(* Logix 5000 project; controller STAT 1756-L72 rev 20.12; software revision 20.04; part 9 of 34 *)
(* tags used below, declared in another part *)
   B14 : DINT[30];
   B16 : DINT[30];
   B17 : DINT[30];
   B3 : DINT[256];
   DateTime : DINT[7];   // DINT array tag for retrieve wallclock time through GSV created during conversion
   I10_000_Bit07 : ALIAS FOR I10[0].7;   // Hand Automaat CL8
   I10_000_Bit10 : ALIAS FOR I10[0].10;   // Drukknop start CL8 PM1
   I10_000_Bit11 : ALIAS FOR I10[0].11;   // Drukknop stop CL8 PM1
   I10_000_Bit12 : ALIAS FOR I10[0].12;   // Drukknop start CL8 PM2
   I10_000_Bit13 : ALIAS FOR I10[0].13;   // Drukknop stop CL8 PM2
   I10_000_Bit14 : ALIAS FOR I10[0].14;   // Drukknop start CL8 PM3
   I10_000_Bit15 : ALIAS FOR I10[0].15;   // Drukknop stop CL8 PM3
   I10_001_Bit00 : ALIAS FOR I10[1].0;   // Drukknop start CL8 PM4
   I10_001_Bit01 : ALIAS FOR I10[1].1;   // Drukknop stop CL8 PM4
   I1_016_Bit02 : ALIAS FOR I1[16].2;   // CL2 start p11
   I1_016_Bit03 : ALIAS FOR I1[16].3;   // CL2 stop p11
   I1_016_Bit04 : ALIAS FOR I1[16].4;   // CL2 start p12
   I1_016_Bit05 : ALIAS FOR I1[16].5;   // CL2 stop p12
   I1_016_Bit11 : ALIAS FOR I1[16].11;   // Niveau lus5 kontakt1
   I1_016_Bit12 : ALIAS FOR I1[16].12;   // Niveau lus5 kontakt2
   I1_017_Bit02 : ALIAS FOR I1[17].2;   // CL3 start p13
   I1_017_Bit03 : ALIAS FOR I1[17].3;   // CL3 stop p13
   I1_017_Bit04 : ALIAS FOR I1[17].4;   // CL3 start p14
   I1_017_Bit05 : ALIAS FOR I1[17].5;   // CL3 stop p14
   I1_017_Bit11 : ALIAS FOR I1[17].11;   // Niveau lus6 kontakt1
   I1_017_Bit12 : ALIAS FOR I1[17].12;   // Niveau lus6 kontakt2
   I1_018_Bit02 : ALIAS FOR I1[18].2;   // CL4 start p15
   I1_018_Bit03 : ALIAS FOR I1[18].3;   // CL4 stop p15
   I1_018_Bit04 : ALIAS FOR I1[18].4;   // CL4 start p16
   I1_018_Bit05 : ALIAS FOR I1[18].5;   // CL4 stop p16
   I1_018_Bit11 : ALIAS FOR I1[18].11;   // Niveau lus7 kontakt1
   I1_018_Bit12 : ALIAS FOR I1[18].12;   // Niveau lus7 kontakt2
   I1_018_Bit13 : ALIAS FOR I1[18].13;   // Niveau lus7 kontakt3
   I2_000_Bit00 : ALIAS FOR I2[0].0;   // Deelnoodstop cl2 lijn 1
   I2_000_Bit01 : ALIAS FOR I2[0].1;   // Deelnoodstop cl3 lijn 3
   I2_000_Bit02 : ALIAS FOR I2[0].2;   // Deelnoodstop cl4
   I2_000_Bit03 : ALIAS FOR I2[0].3;   // Deelnoodstop cl5 lijn 4
   I2_000_Bit06 : ALIAS FOR I2[0].6;   // Deelnoodstop cl7 IBT B
   I6_001_Bit12 : ALIAS FOR I6[1].12;   // Ph meting vervuild water fout
   I7_000_Bit01 : ALIAS FOR I7[0].1;   // lus2 niveau kontakt 1
   I7_000_Bit04 : ALIAS FOR I7[0].4;   // lus3 niveau kontakt 1
   I7_000_Bit10 : ALIAS FOR I7[0].10;   // zeer hoog alarm ketel clarifee
   I7_001_Bit13 : ALIAS FOR I7[1].13;   // lus 8 niveau kontakt 1
   I7_001_Bit14 : ALIAS FOR I7[1].14;   // lus 8 niveau kontakt 2
   I7_001_Bit15 : ALIAS FOR I7[1].15;   // lus 8 niveau kontakt 3
   I8_001_Bit01 : ALIAS FOR I8[1].1;   // hand automaat cl5
   I8_001_Bit02 : ALIAS FOR I8[1].2;   // drukknop start cl5 p17
   I8_001_Bit03 : ALIAS FOR I8[1].3;   // drukknop stop cl5 p17
   I8_001_Bit04 : ALIAS FOR I8[1].4;   // drukknop start cl5 p18
   I8_001_Bit05 : ALIAS FOR I8[1].5;   // drukknop stop cl5 p18
   I9_000_Bit09 : ALIAS FOR I9[0].9;   // Hand_Auto CL7
   I9_001_Bit12 : ALIAS FOR I9[1].12;   // Drukknop start CL7 A
   I9_001_Bit13 : ALIAS FOR I9[1].13;   // Drukknop stop CL7 pd7
   I9_001_Bit14 : ALIAS FOR I9[1].14;   // drukknop start cl7 pd8
   I9_001_Bit15 : ALIAS FOR I9[1].15;   // drukknop stop cl7 pd8
   N11 : DINT[150];
   N12 : DINT[230];
   N13 : DINT[230];
   N20 : DINT[80];
   N21 : DINT[80];
   O12_000_Bit04 : ALIAS FOR O12[0].4;   // Motor doseerpomp acide pd3 PD3_DOS_ACIDE
   O12_000_Bit05 : ALIAS FOR O12[0].5;   // Motor doseerpomp acide pd4 PD4_DOS_ACIDE
   O12_000_Bit06 : ALIAS FOR O12[0].6;   // Motor doseerpomp acide pd5 soude PD5_DOS_SOUDE
   O12_000_Bit07 : ALIAS FOR O12[0].7;   // Motor doseerpomp acide pd6 soude PD6_DOS_SOUDE
   O12_000_Bit10 : ALIAS FOR O12[0].10;   // pomp pd7 doseerpomp floculaat PD7_DOSEER_FLOCU
   O12_000_Bit11 : ALIAS FOR O12[0].11;   // pomp pd8 doseerpomp floculaat PD8_DOSEER_FLOCU
   O12_000_Bit14 : ALIAS FOR O12[0].14;   // Motor Pm1 recerculatiepomp ingang 1 decanter PM1_RECER_DEC1
   O12_000_Bit15 : ALIAS FOR O12[0].15;   // Motor Pm2 recerculatiepomp ingang 2 decanter PM2_RECER_DEC2
   O12_001_Bit00 : ALIAS FOR O12[1].0;   // Motor Pm3 evacuatiepomp ingang 1 decanter PM3_EVACU_IN_1
   O12_001_Bit01 : ALIAS FOR O12[1].1;   // Motor Pm4 evacuatiepomp ingang 2 decanter PM4_EVACU_IN_2
   O13_000_Bit06 : ALIAS FOR O13[0].6;   // PULS_DOSEER_PD3
   O13_000_Bit07 : ALIAS FOR O13[0].7;   // PULS_DOSEER_PD4
   O13_000_Bit08 : ALIAS FOR O13[0].8;   // PULS_DOSEER_PD5
   O13_000_Bit09 : ALIAS FOR O13[0].9;   // PULS_DOSEER_PD6
   O15_001_Bit07 : ALIAS FOR O15[1].7;   // EV3 EV3
   O15_001_Bit08 : ALIAS FOR O15[1].8;   // EV4 EV4
   O15_001_Bit09 : ALIAS FOR O15[1].9;   // EV5 EV5
   P11_RECUP : BOOL;
   P13_RECUP : BOOL;
   P14_RECUP : BOOL;
   p15 : BOOL;
   P16 : BOOL;
   P17 : BOOL;
   P18 : BOOL;
   pd3 : BOOL;
   pd4 : BOOL;
   pd5 : BOOL;
   pd6 : BOOL;
   PD7 : BOOL;
   PD8 : BOOL;
   PM1 : BOOL;
   PM2 : BOOL;
   PM3 : BOOL;
   PM4 : BOOL;
   PMP_L1_ET_L3_RUN : BOOL;
   POS_EV3 : BOOL;
   T27 : TIMER[100];
   T4 : TIMER[200];
(* ibt, continued *)

ROUTINE _11_PM1_PM4   (* ladder *)
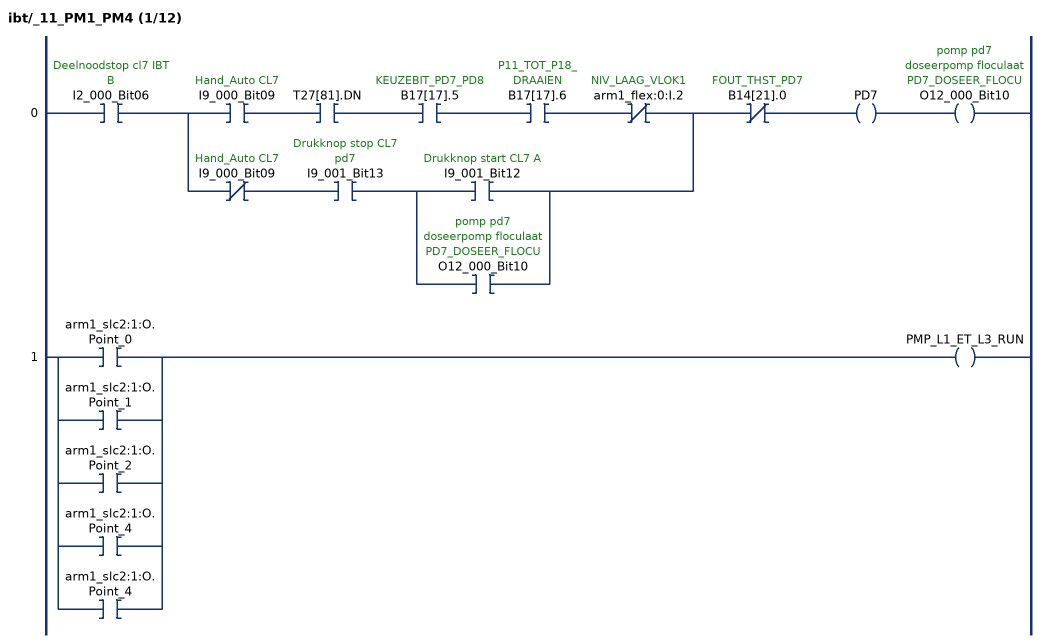
   0: XIC(I2_000_Bit06)[XIC(I9_000_Bit09) XIC(T27[81].DN) XIC(B17[17].5) XIC(B17[17].6) XIO(arm1_flex:0:I.2) ,XIO(I9_000_Bit09) XIC(I9_001_Bit13) [XIC(I9_001_Bit12) ,XIC(O12_000_Bit10) ] ]XIO(B14[21].0)OTE(PD7)OTE(O12_000_Bit10);
   1: [XIC(arm1_slc2:1:O.Point_0) ,[XIC(arm1_slc2:1:O.Point_1) ,[XIC(arm1_slc2:1:O.Point_2) ,[XIC(arm1_slc2:1:O.Point_4) ,XIC(arm1_slc2:1:O.Point_4) ] ] ] ]OTE(PMP_L1_ET_L3_RUN);
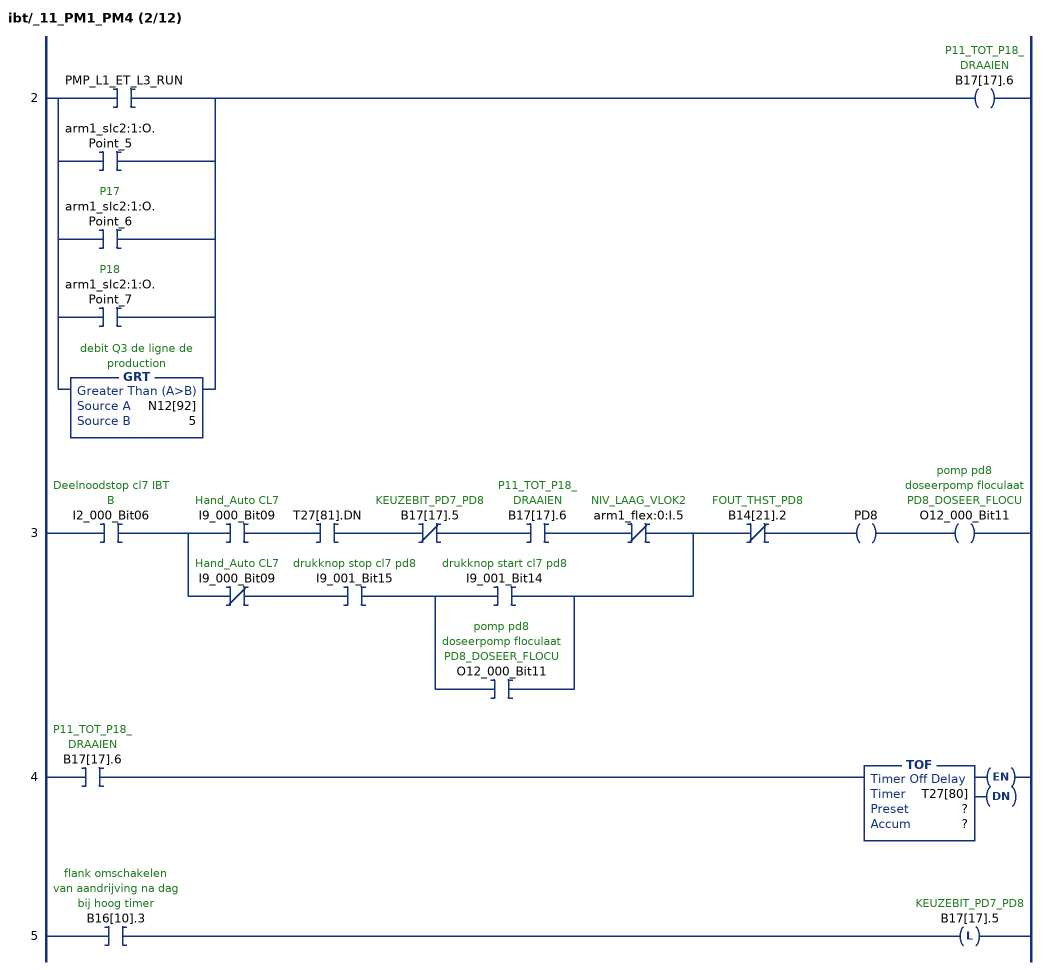
   2: [XIC(PMP_L1_ET_L3_RUN) ,[XIC(arm1_slc2:1:O.Point_5) ,[XIC(arm1_slc2:1:O.Point_6) ,[XIC(arm1_slc2:1:O.Point_7) ,GRT(N12[92],5) ] ] ] ]OTE(B17[17].6);
   3: XIC(I2_000_Bit06)[XIC(I9_000_Bit09) XIC(T27[81].DN) XIO(B17[17].5) XIC(B17[17].6) XIO(arm1_flex:0:I.5) ,XIO(I9_000_Bit09) XIC(I9_001_Bit15) [XIC(I9_001_Bit14) ,XIC(O12_000_Bit11) ] ]XIO(B14[21].2)OTE(PD8)OTE(O12_000_Bit11);
   4: XIC(B17[17].6)TOF(T27[80],?,?);
   5: XIC(B16[10].3)OTL(B17[17].5);
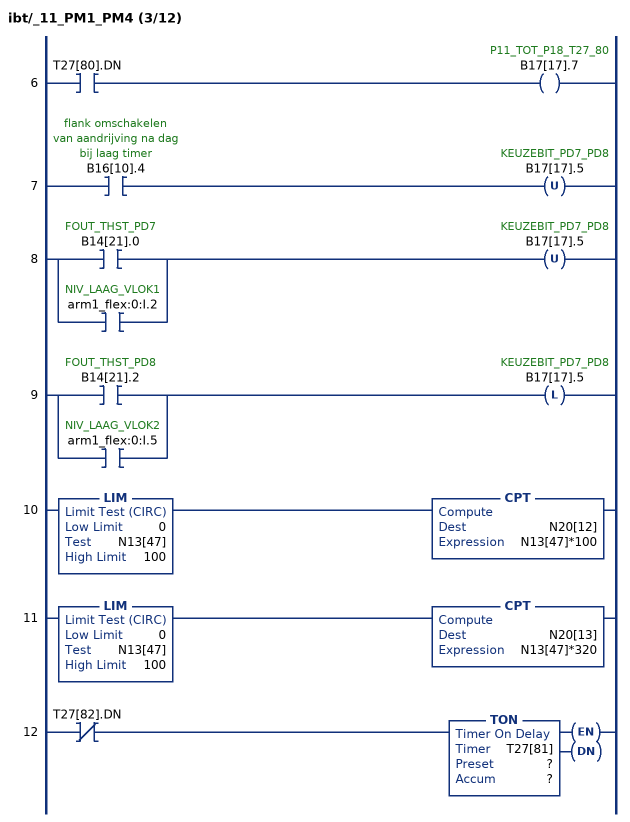
   6: XIC(T27[80].DN)OTE(B17[17].7);
   7: XIC(B16[10].4)OTU(B17[17].5);
   8: [XIC(B14[21].0) ,XIC(arm1_flex:0:I.2) ]OTU(B17[17].5);
   9: [XIC(B14[21].2) ,XIC(arm1_flex:0:I.5) ]OTL(B17[17].5);
   10: LIM(0,N13[47],100)CPT(N20[12],N13[47]*100);
   11: LIM(0,N13[47],100)CPT(N20[13],N13[47]*320);
   12: XIO(T27[82].DN)TON(T27[81],?,?);
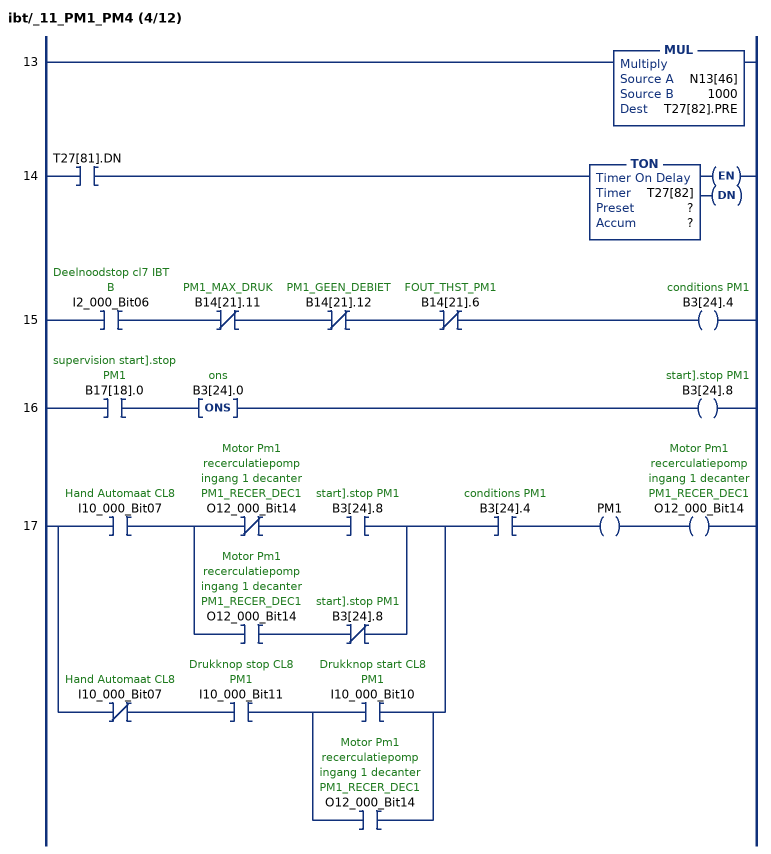
   13: MUL(N13[46],1000,T27[82].PRE);
   14: XIC(T27[81].DN)TON(T27[82],?,?);
   15: XIC(I2_000_Bit06)XIO(B14[21].11)XIO(B14[21].12)XIO(B14[21].6)OTE(B3[24].4);
   16: XIC(B17[18].0)ONS(B3[24].0)OTE(B3[24].8);
   17: [XIC(I10_000_Bit07) [XIO(O12_000_Bit14) XIC(B3[24].8) ,XIC(O12_000_Bit14) XIO(B3[24].8) ] ,XIO(I10_000_Bit07) XIC(I10_000_Bit11) [XIC(I10_000_Bit10) ,XIC(O12_000_Bit14) ] ]XIC(B3[24].4)OTE(PM1)OTE(O12_000_Bit14);
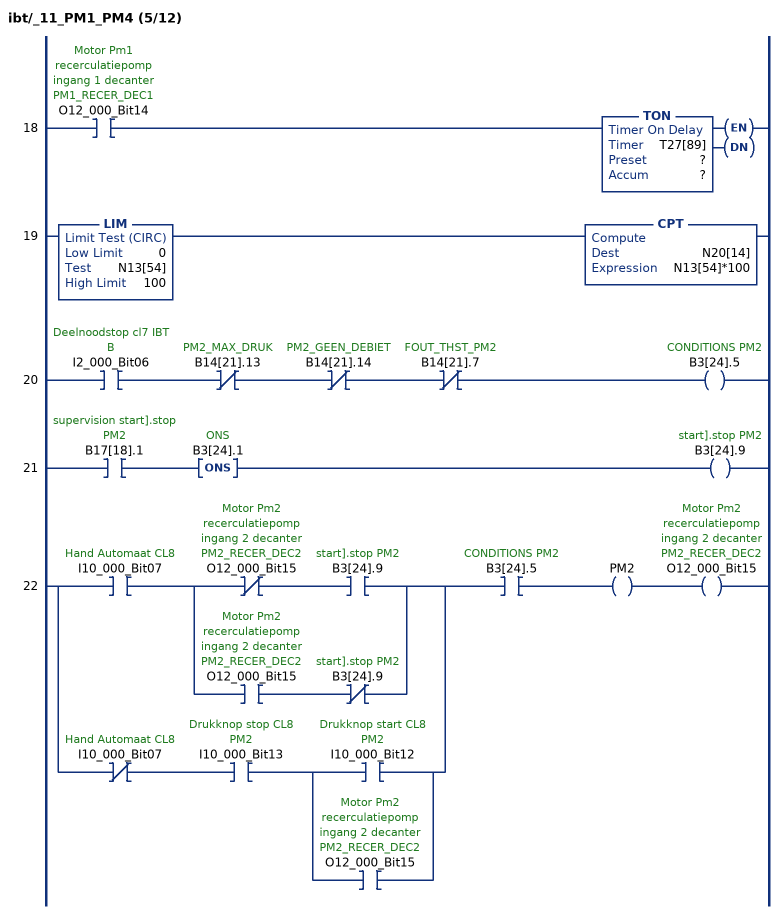
   18: XIC(O12_000_Bit14)TON(T27[89],?,?);
   19: LIM(0,N13[54],100)CPT(N20[14],N13[54]*100);
   20: XIC(I2_000_Bit06)XIO(B14[21].13)XIO(B14[21].14)XIO(B14[21].7)OTE(B3[24].5);
   21: XIC(B17[18].1)ONS(B3[24].1)OTE(B3[24].9);
   22: [XIC(I10_000_Bit07) [XIO(O12_000_Bit15) XIC(B3[24].9) ,XIC(O12_000_Bit15) XIO(B3[24].9) ] ,XIO(I10_000_Bit07) XIC(I10_000_Bit13) [XIC(I10_000_Bit12) ,XIC(O12_000_Bit15) ] ]XIC(B3[24].5)OTE(PM2)OTE(O12_000_Bit15);
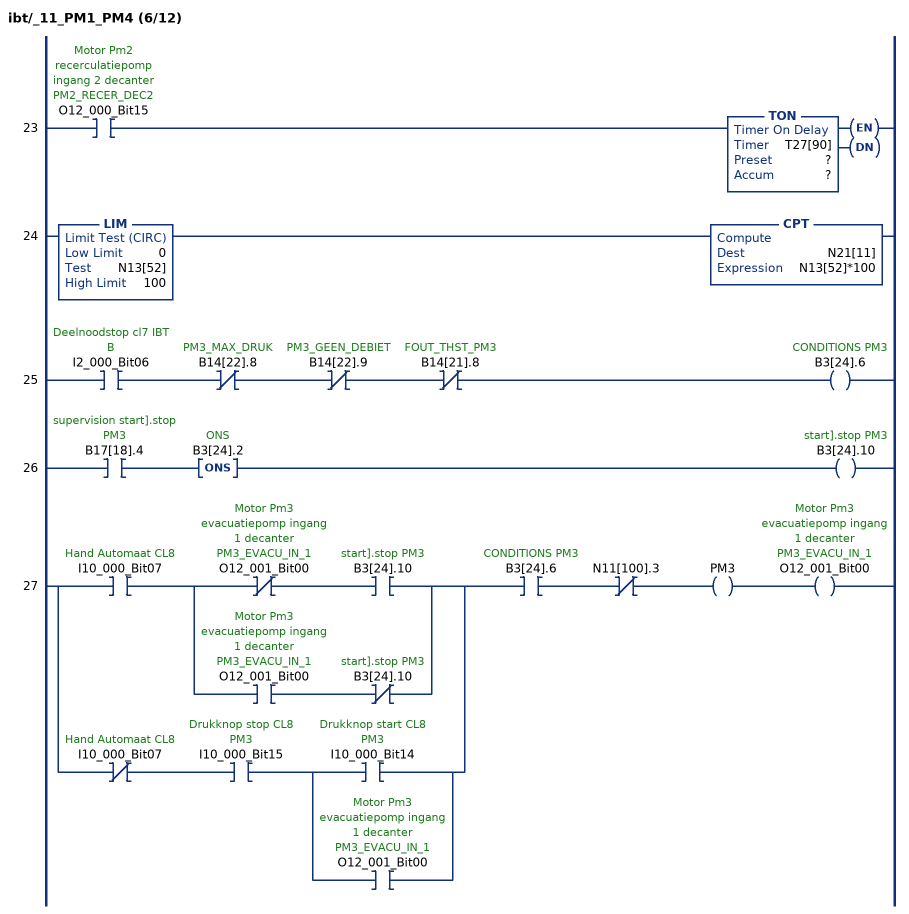
   23: XIC(O12_000_Bit15)TON(T27[90],?,?);
   24: LIM(0,N13[52],100)CPT(N21[11],N13[52]*100);
   25: XIC(I2_000_Bit06)XIO(B14[22].8)XIO(B14[22].9)XIO(B14[21].8)OTE(B3[24].6);
   26: XIC(B17[18].4)ONS(B3[24].2)OTE(B3[24].10);
   27: [XIC(I10_000_Bit07) [XIO(O12_001_Bit00) XIC(B3[24].10) ,XIC(O12_001_Bit00) XIO(B3[24].10) ] ,XIO(I10_000_Bit07) XIC(I10_000_Bit15) [XIC(I10_000_Bit14) ,XIC(O12_001_Bit00) ] ]XIC(B3[24].6)XIO(N11[100].3)OTE(PM3)OTE(O12_001_Bit00);
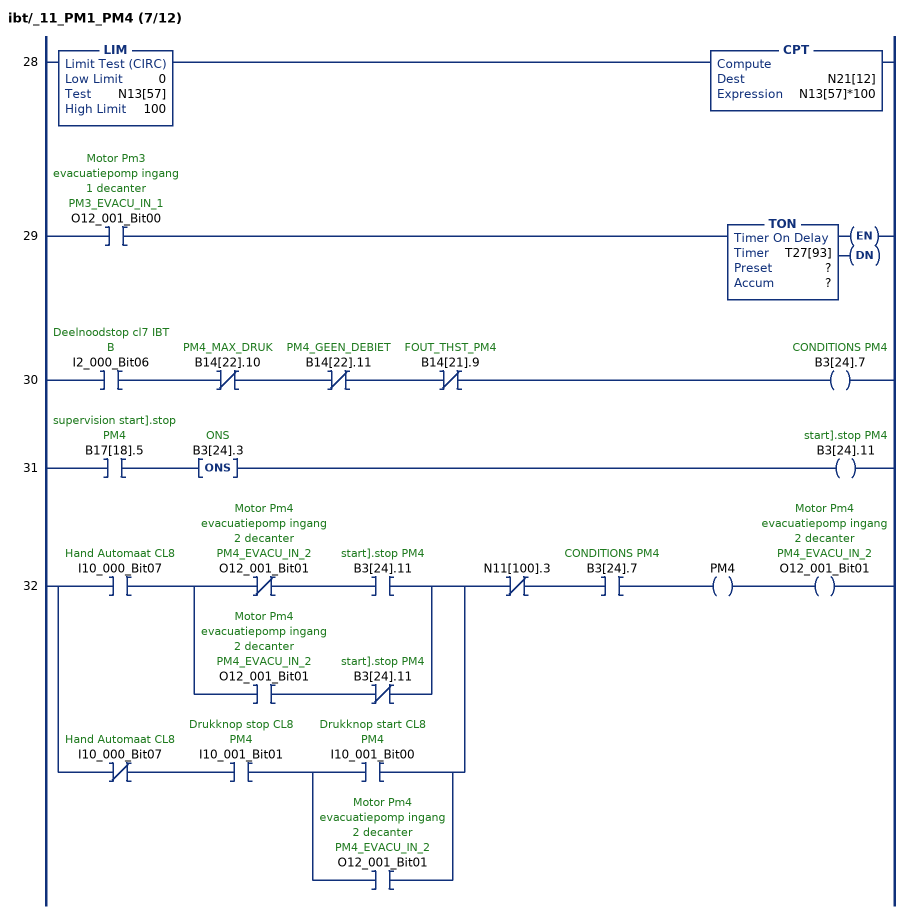
   28: LIM(0,N13[57],100)CPT(N21[12],N13[57]*100);
   29: XIC(O12_001_Bit00)TON(T27[93],?,?);
   30: XIC(I2_000_Bit06)XIO(B14[22].10)XIO(B14[22].11)XIO(B14[21].9)OTE(B3[24].7);
   31: XIC(B17[18].5)ONS(B3[24].3)OTE(B3[24].11);
   32: [XIC(I10_000_Bit07) [XIO(O12_001_Bit01) XIC(B3[24].11) ,XIC(O12_001_Bit01) XIO(B3[24].11) ] ,XIO(I10_000_Bit07) XIC(I10_001_Bit01) [XIC(I10_001_Bit00) ,XIC(O12_001_Bit01) ] ]XIO(N11[100].3)XIC(B3[24].7)OTE(PM4)OTE(O12_001_Bit01);
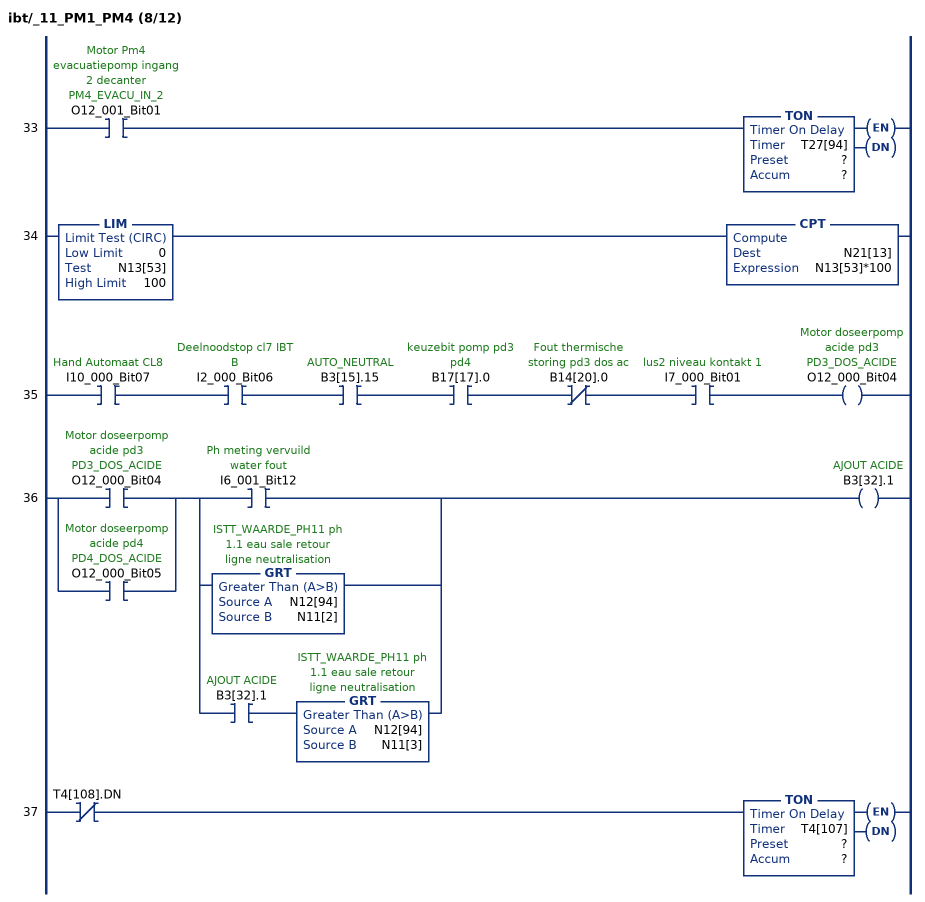
   33: XIC(O12_001_Bit01)TON(T27[94],?,?);
   34: LIM(0,N13[53],100)CPT(N21[13],N13[53]*100);
   35: XIC(I10_000_Bit07)XIC(I2_000_Bit06)XIC(B3[15].15)XIC(B17[17].0)XIO(B14[20].0)XIC(I7_000_Bit01)OTE(O12_000_Bit04);
   36: [XIC(O12_000_Bit04) ,XIC(O12_000_Bit05) ][XIC(I6_001_Bit12) ,GRT(N12[94],N11[2]) ,XIC(B3[32].1) GRT(N12[94],N11[3]) ]OTE(B3[32].1);
   37: XIO(T4[108].DN)TON(T4[107],?,?);
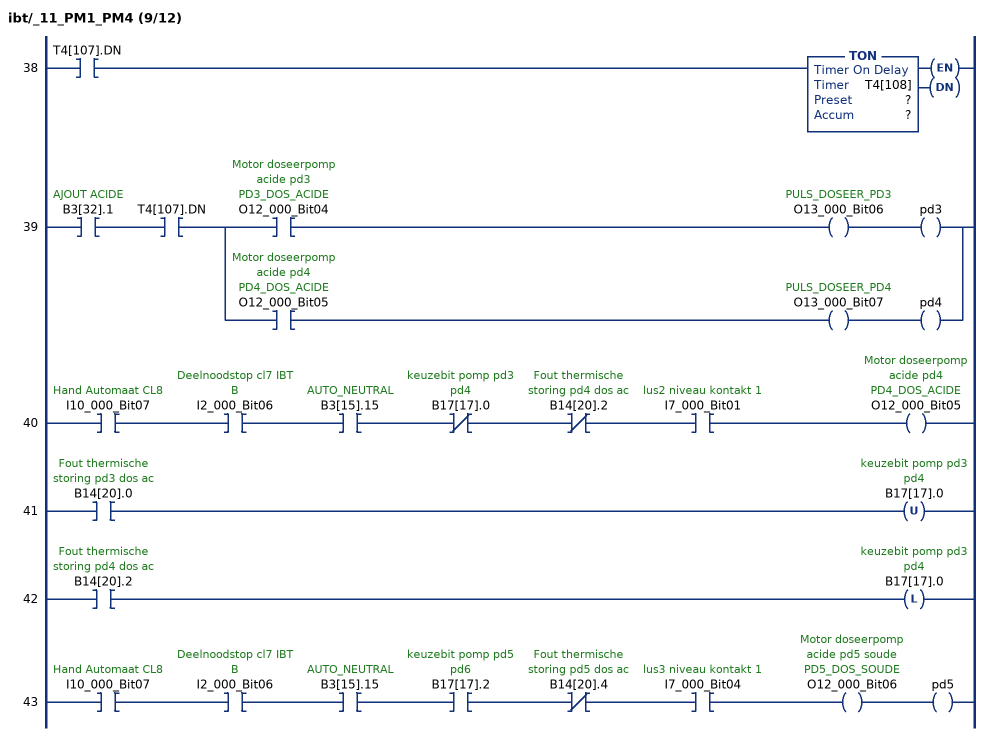
   38: XIC(T4[107].DN)TON(T4[108],?,?);
   39: XIC(B3[32].1)XIC(T4[107].DN)[XIC(O12_000_Bit04) OTE(O13_000_Bit06) OTE(pd3) ,XIC(O12_000_Bit05) OTE(O13_000_Bit07) OTE(pd4) ];
   40: XIC(I10_000_Bit07)XIC(I2_000_Bit06)XIC(B3[15].15)XIO(B17[17].0)XIO(B14[20].2)XIC(I7_000_Bit01)OTE(O12_000_Bit05);
   41: XIC(B14[20].0)OTU(B17[17].0);
   42: XIC(B14[20].2)OTL(B17[17].0);
   43: XIC(I10_000_Bit07)XIC(I2_000_Bit06)XIC(B3[15].15)XIC(B17[17].2)XIO(B14[20].4)XIC(I7_000_Bit04)OTE(O12_000_Bit06)OTE(pd5);
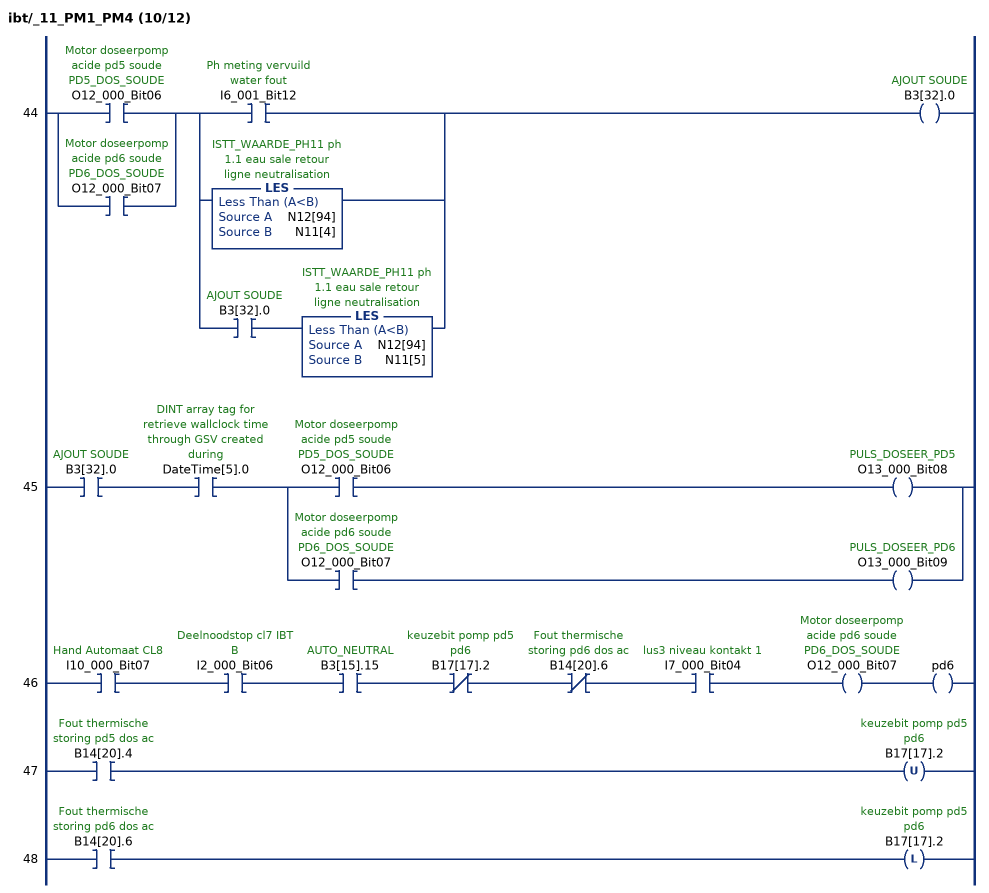
   44: [XIC(O12_000_Bit06) ,XIC(O12_000_Bit07) ][XIC(I6_001_Bit12) ,LES(N12[94],N11[4]) ,XIC(B3[32].0) LES(N12[94],N11[5]) ]OTE(B3[32].0);
   45: XIC(B3[32].0)XIC(DateTime[5].0)[XIC(O12_000_Bit06) OTE(O13_000_Bit08) ,XIC(O12_000_Bit07) OTE(O13_000_Bit09) ];
   46: XIC(I10_000_Bit07)XIC(I2_000_Bit06)XIC(B3[15].15)XIO(B17[17].2)XIO(B14[20].6)XIC(I7_000_Bit04)OTE(O12_000_Bit07)OTE(pd6);
   47: XIC(B14[20].4)OTU(B17[17].2);
   48: XIC(B14[20].6)OTL(B17[17].2);
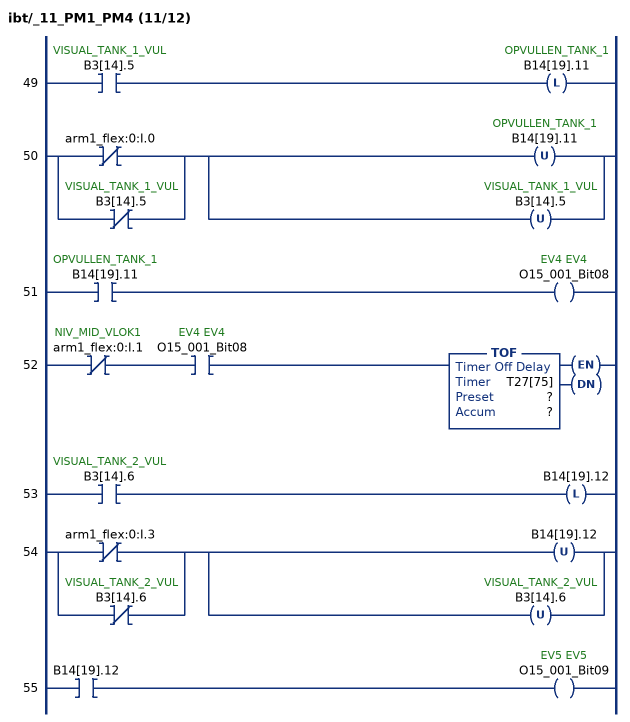
   49: XIC(B3[14].5)OTL(B14[19].11);
   50: [XIO(arm1_flex:0:I.0) ,XIO(B3[14].5) ][OTU(B14[19].11) ,OTU(B3[14].5) ];
   51: XIC(B14[19].11)OTE(O15_001_Bit08);
   52: XIO(arm1_flex:0:I.1)XIC(O15_001_Bit08)TOF(T27[75],?,?);
   53: XIC(B3[14].6)OTL(B14[19].12);
   54: [XIO(arm1_flex:0:I.3) ,XIO(B3[14].6) ][OTU(B14[19].12) ,OTU(B3[14].6) ];
   55: XIC(B14[19].12)OTE(O15_001_Bit09);
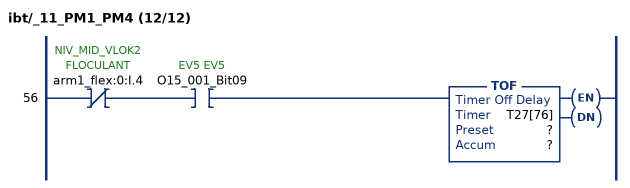
   56: XIO(arm1_flex:0:I.4)XIC(O15_001_Bit09)TOF(T27[76],?,?);
END_ROUTINE

ROUTINE _12_P11_P18   (* ladder *)
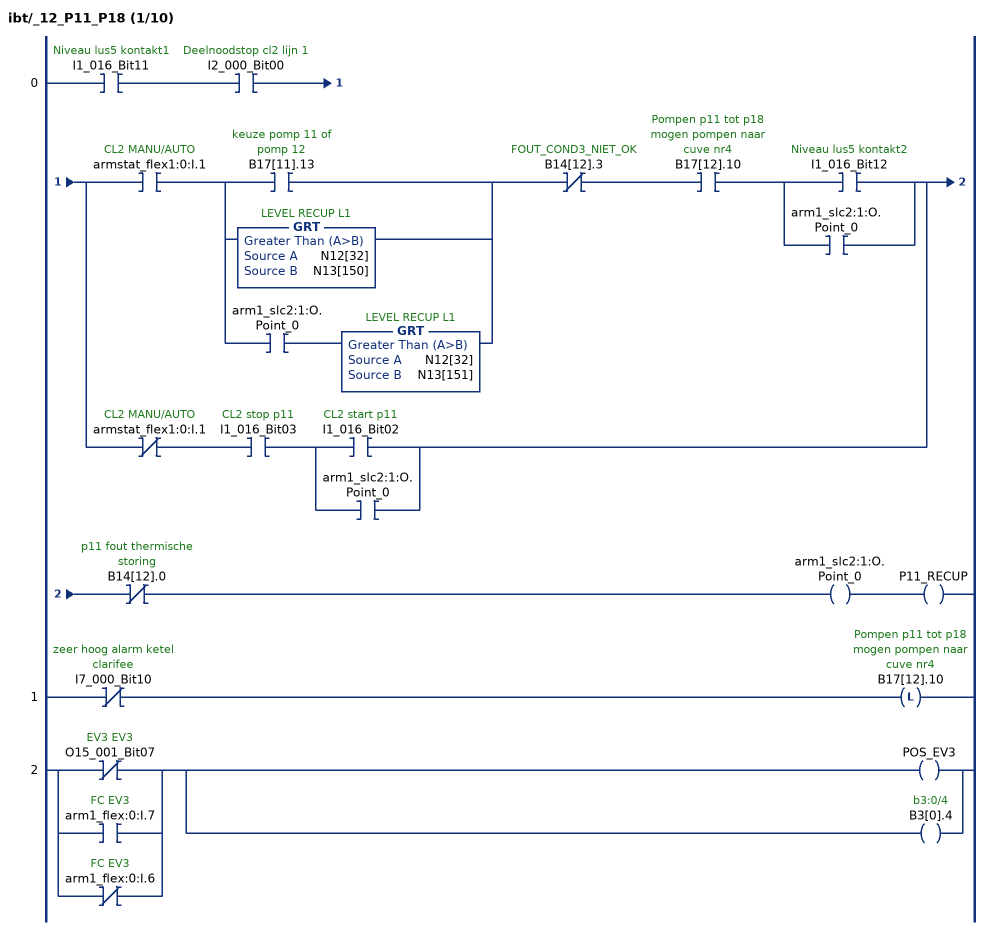
   0: XIC(I1_016_Bit11)XIC(I2_000_Bit00)[XIC(armstat_flex1:0:I.1) [XIC(B17[11].13) ,GRT(N12[32],N13[150]) ,XIC(arm1_slc2:1:O.Point_0) GRT(N12[32],N13[151]) ] XIO(B14[12].3) XIC(B17[12].10) [XIC(I1_016_Bit12) ,XIC(arm1_slc2:1:O.Point_0) ] ,XIO(armstat_flex1:0:I.1) XIC(I1_016_Bit03) [XIC(I1_016_Bit02) ,XIC(arm1_slc2:1:O.Point_0) ] ]XIO(B14[12].0)OTE(arm1_slc2:1:O.Point_0)OTE(P11_RECUP);
   1: XIO(I7_000_Bit10)OTL(B17[12].10);
   2: [XIO(O15_001_Bit07) ,[XIC(arm1_flex:0:I.7) ,XIO(arm1_flex:0:I.6) ] ][OTE(POS_EV3) ,OTE(B3[0].4) ];
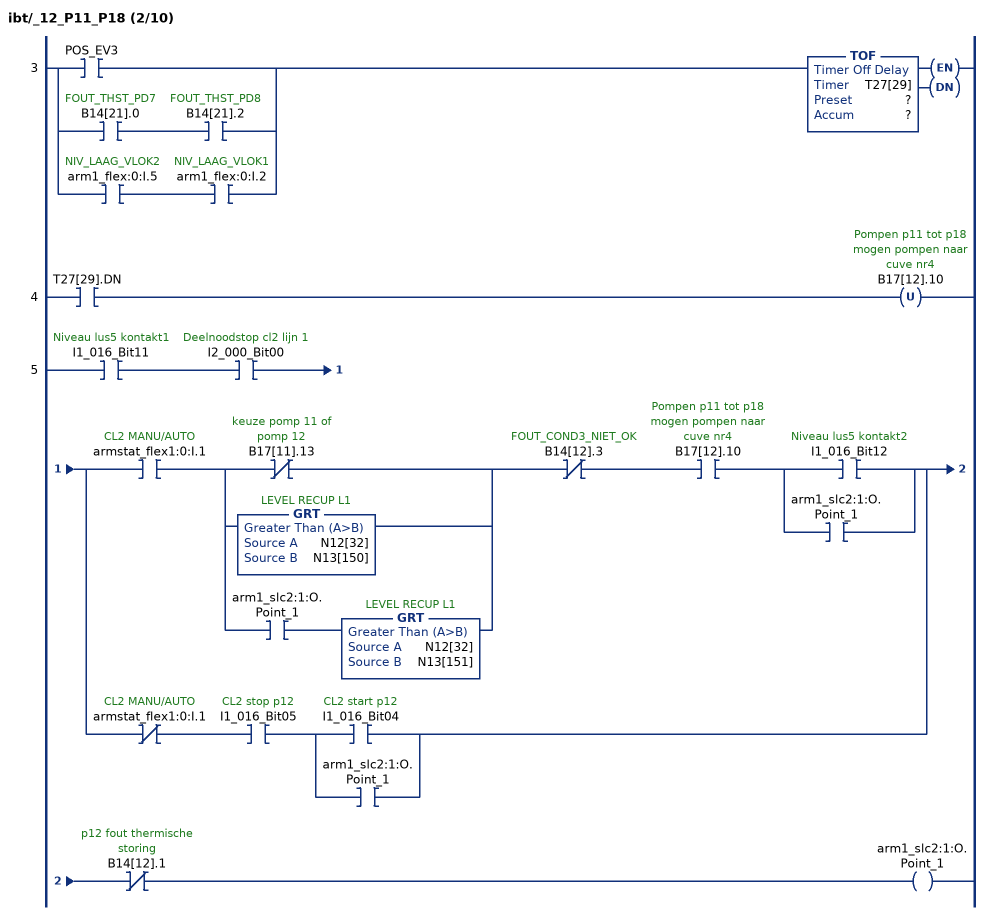
   3: [XIC(POS_EV3) ,XIC(B14[21].0) XIC(B14[21].2) ,XIC(arm1_flex:0:I.5) XIC(arm1_flex:0:I.2) ]TOF(T27[29],?,?);
   4: XIC(T27[29].DN)OTU(B17[12].10);
   5: XIC(I1_016_Bit11)XIC(I2_000_Bit00)[XIC(armstat_flex1:0:I.1) [XIO(B17[11].13) ,GRT(N12[32],N13[150]) ,XIC(arm1_slc2:1:O.Point_1) GRT(N12[32],N13[151]) ] XIO(B14[12].3) XIC(B17[12].10) [XIC(I1_016_Bit12) ,XIC(arm1_slc2:1:O.Point_1) ] ,XIO(armstat_flex1:0:I.1) XIC(I1_016_Bit05) [XIC(I1_016_Bit04) ,XIC(arm1_slc2:1:O.Point_1) ] ]XIO(B14[12].1)OTE(arm1_slc2:1:O.Point_1);
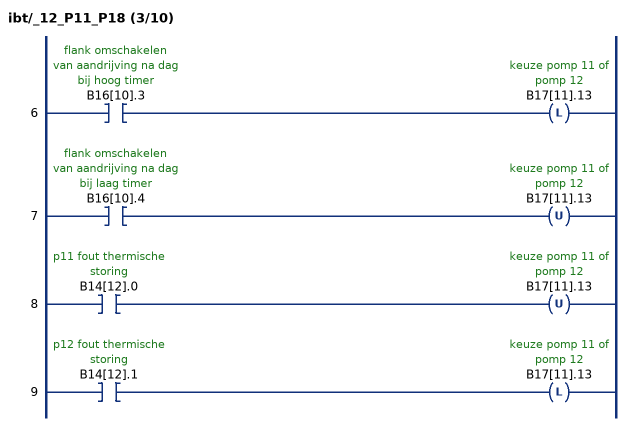
   6: XIC(B16[10].3)OTL(B17[11].13);
   7: XIC(B16[10].4)OTU(B17[11].13);
   8: XIC(B14[12].0)OTU(B17[11].13);
   9: XIC(B14[12].1)OTL(B17[11].13);
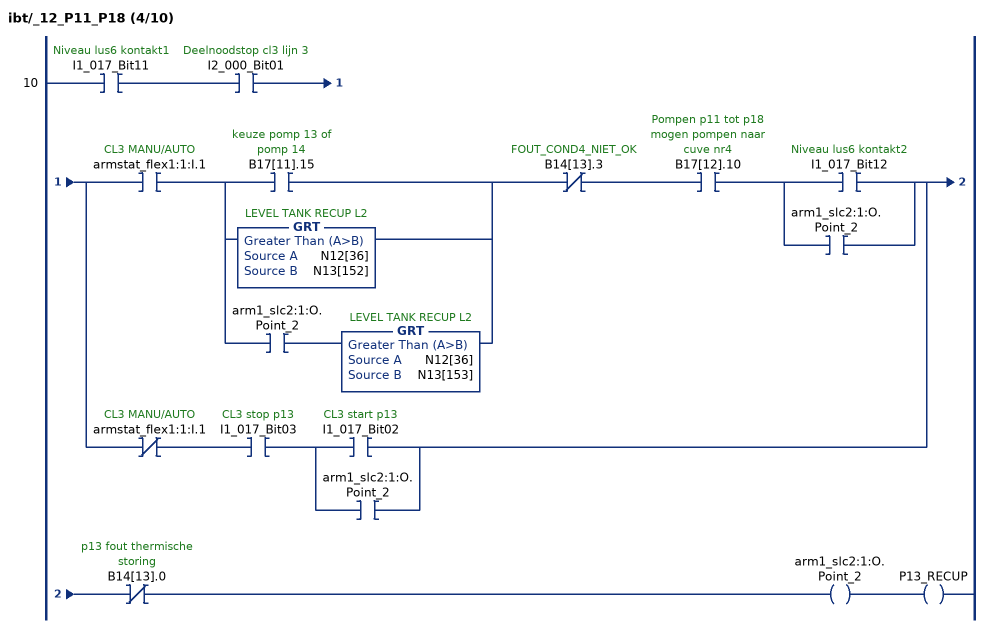
   10: XIC(I1_017_Bit11)XIC(I2_000_Bit01)[XIC(armstat_flex1:1:I.1) [XIC(B17[11].15) ,GRT(N12[36],N13[152]) ,XIC(arm1_slc2:1:O.Point_2) GRT(N12[36],N13[153]) ] XIO(B14[13].3) XIC(B17[12].10) [XIC(I1_017_Bit12) ,XIC(arm1_slc2:1:O.Point_2) ] ,XIO(armstat_flex1:1:I.1) XIC(I1_017_Bit03) [XIC(I1_017_Bit02) ,XIC(arm1_slc2:1:O.Point_2) ] ]XIO(B14[13].0)OTE(arm1_slc2:1:O.Point_2)OTE(P13_RECUP);
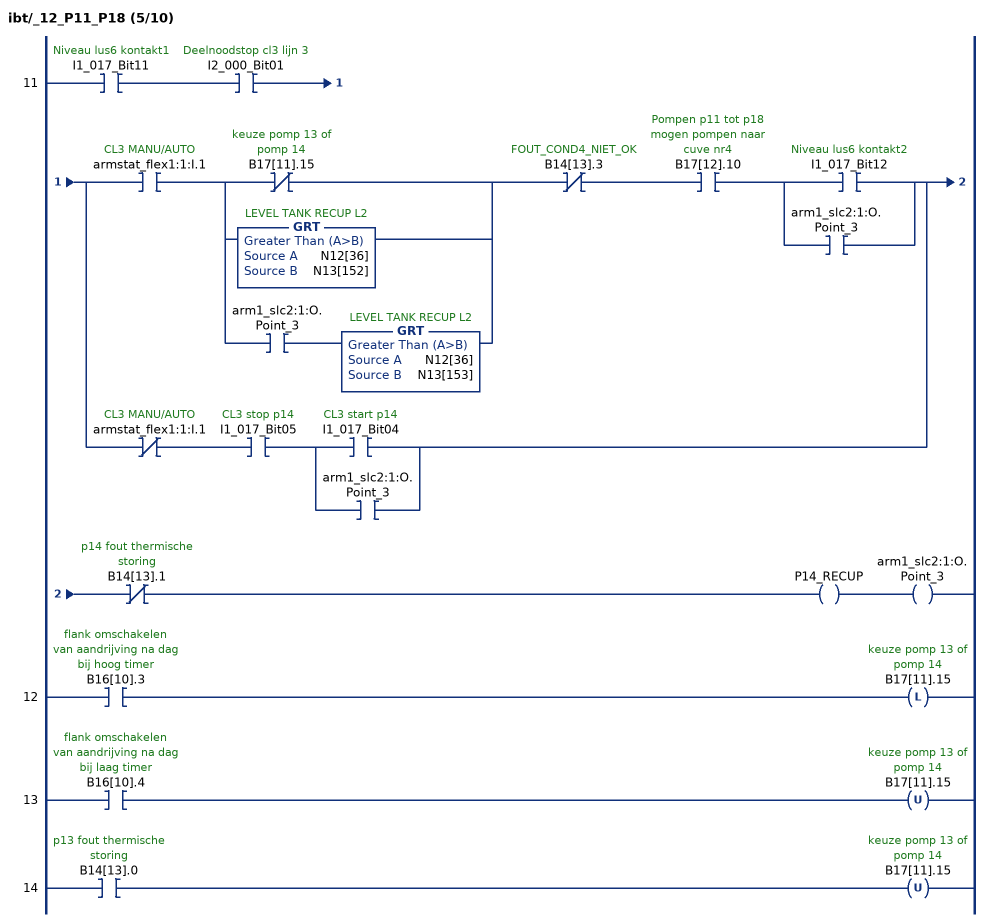
   11: XIC(I1_017_Bit11)XIC(I2_000_Bit01)[XIC(armstat_flex1:1:I.1) [XIO(B17[11].15) ,GRT(N12[36],N13[152]) ,XIC(arm1_slc2:1:O.Point_3) GRT(N12[36],N13[153]) ] XIO(B14[13].3) XIC(B17[12].10) [XIC(I1_017_Bit12) ,XIC(arm1_slc2:1:O.Point_3) ] ,XIO(armstat_flex1:1:I.1) XIC(I1_017_Bit05) [XIC(I1_017_Bit04) ,XIC(arm1_slc2:1:O.Point_3) ] ]XIO(B14[13].1)OTE(P14_RECUP)OTE(arm1_slc2:1:O.Point_3);
   12: XIC(B16[10].3)OTL(B17[11].15);
   13: XIC(B16[10].4)OTU(B17[11].15);
   14: XIC(B14[13].0)OTU(B17[11].15);
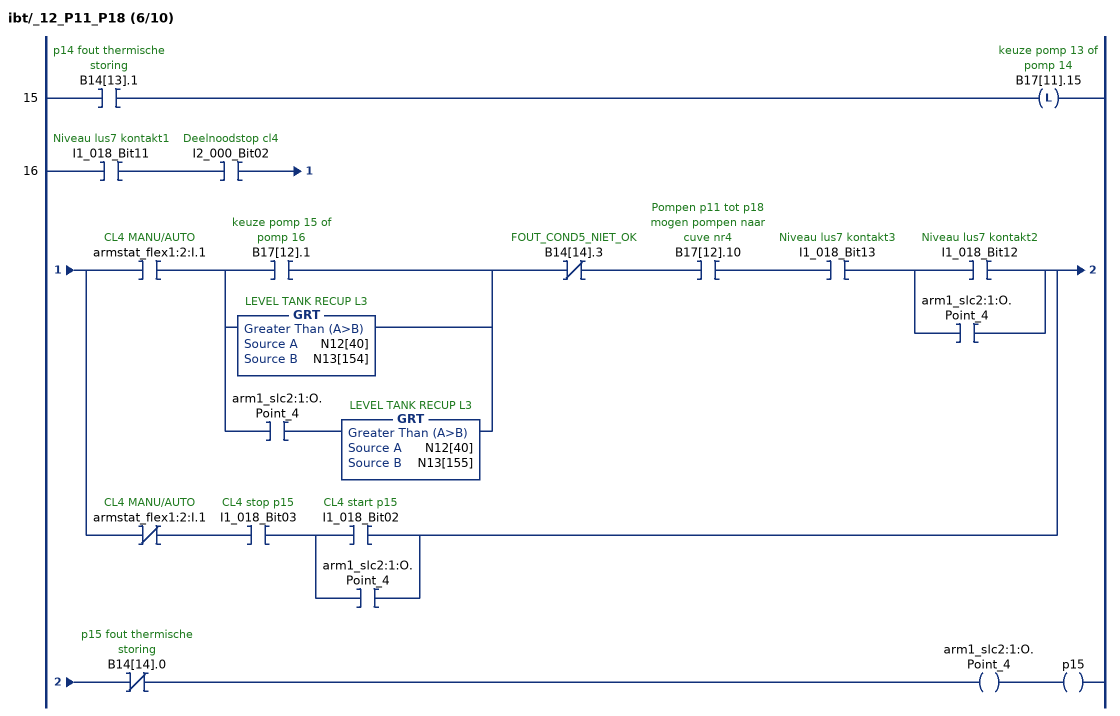
   15: XIC(B14[13].1)OTL(B17[11].15);
   16: XIC(I1_018_Bit11)XIC(I2_000_Bit02)[XIC(armstat_flex1:2:I.1) [XIC(B17[12].1) ,GRT(N12[40],N13[154]) ,XIC(arm1_slc2:1:O.Point_4) GRT(N12[40],N13[155]) ] XIO(B14[14].3) XIC(B17[12].10) XIC(I1_018_Bit13) [XIC(I1_018_Bit12) ,XIC(arm1_slc2:1:O.Point_4) ] ,XIO(armstat_flex1:2:I.1) XIC(I1_018_Bit03) [XIC(I1_018_Bit02) ,XIC(arm1_slc2:1:O.Point_4) ] ]XIO(B14[14].0)OTE(arm1_slc2:1:O.Point_4)OTE(p15);
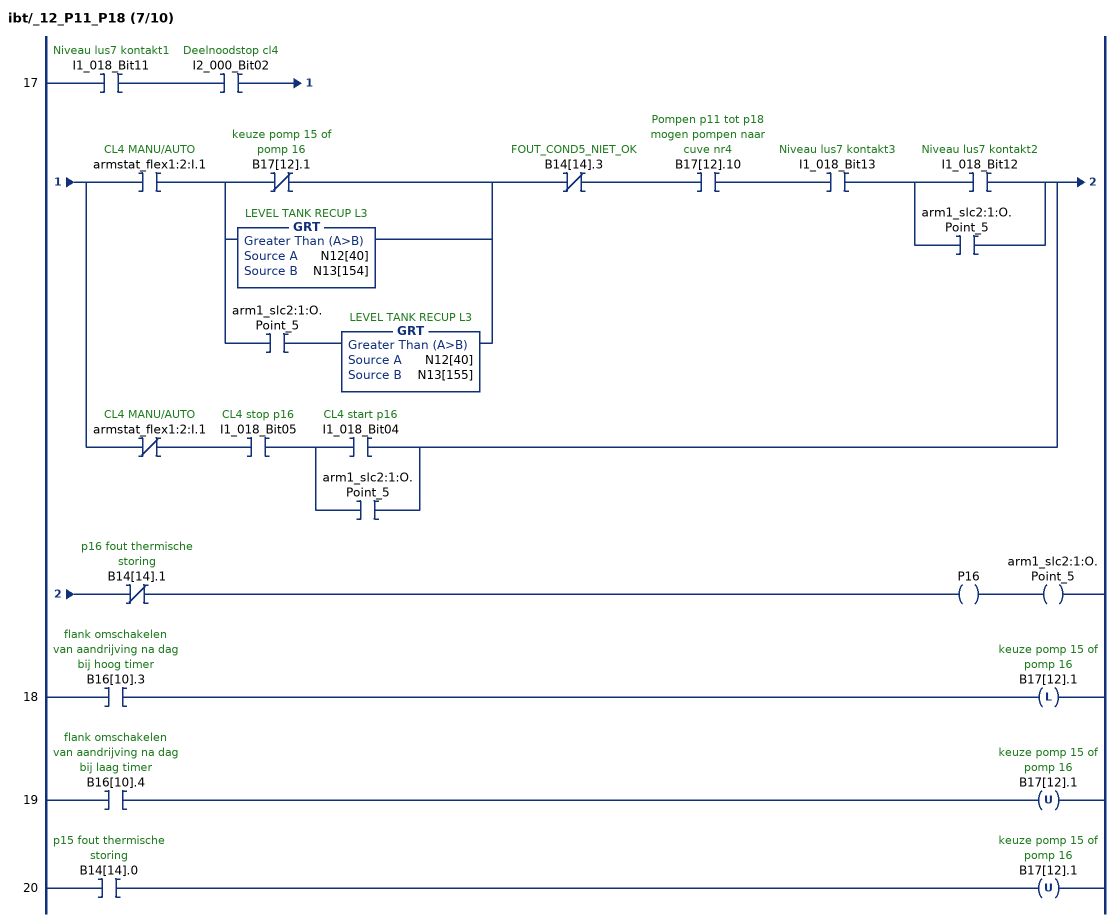
   17: XIC(I1_018_Bit11)XIC(I2_000_Bit02)[XIC(armstat_flex1:2:I.1) [XIO(B17[12].1) ,GRT(N12[40],N13[154]) ,XIC(arm1_slc2:1:O.Point_5) GRT(N12[40],N13[155]) ] XIO(B14[14].3) XIC(B17[12].10) XIC(I1_018_Bit13) [XIC(I1_018_Bit12) ,XIC(arm1_slc2:1:O.Point_5) ] ,XIO(armstat_flex1:2:I.1) XIC(I1_018_Bit05) [XIC(I1_018_Bit04) ,XIC(arm1_slc2:1:O.Point_5) ] ]XIO(B14[14].1)OTE(P16)OTE(arm1_slc2:1:O.Point_5);
   18: XIC(B16[10].3)OTL(B17[12].1);
   19: XIC(B16[10].4)OTU(B17[12].1);
   20: XIC(B14[14].0)OTU(B17[12].1);
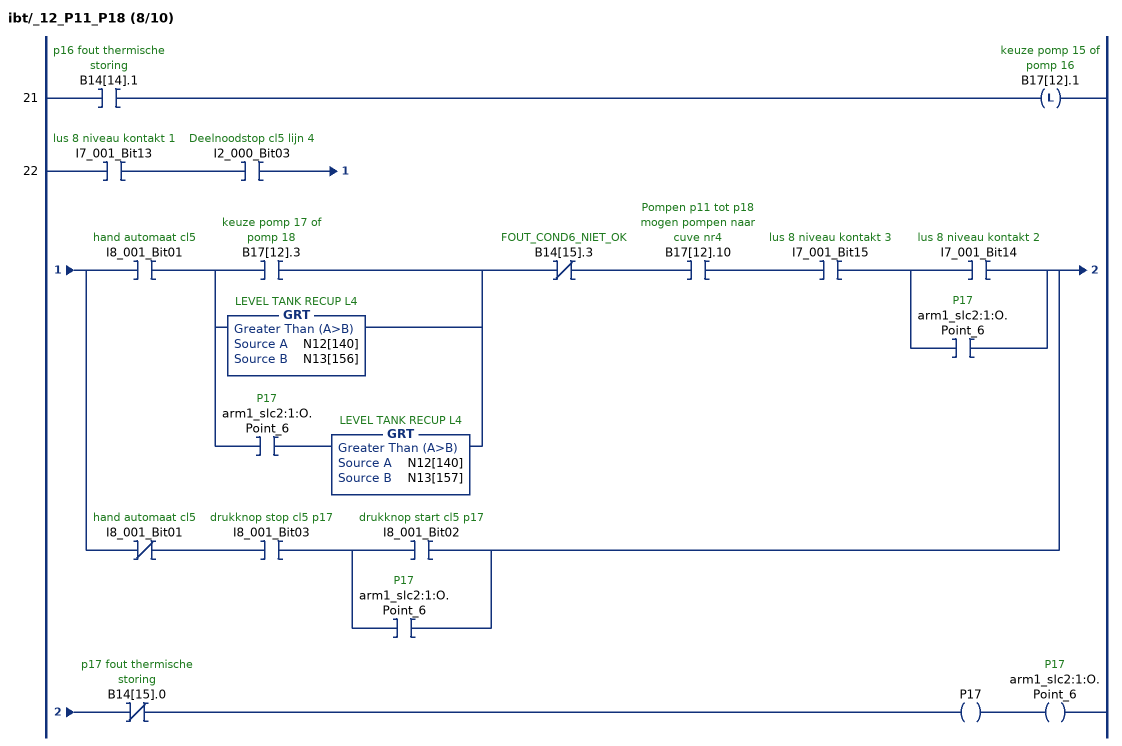
   21: XIC(B14[14].1)OTL(B17[12].1);
   22: XIC(I7_001_Bit13)XIC(I2_000_Bit03)[XIC(I8_001_Bit01) [XIC(B17[12].3) ,GRT(N12[140],N13[156]) ,XIC(arm1_slc2:1:O.Point_6) GRT(N12[140],N13[157]) ] XIO(B14[15].3) XIC(B17[12].10) XIC(I7_001_Bit15) [XIC(I7_001_Bit14) ,XIC(arm1_slc2:1:O.Point_6) ] ,XIO(I8_001_Bit01) XIC(I8_001_Bit03) [XIC(I8_001_Bit02) ,XIC(arm1_slc2:1:O.Point_6) ] ]XIO(B14[15].0)OTE(P17)OTE(arm1_slc2:1:O.Point_6);
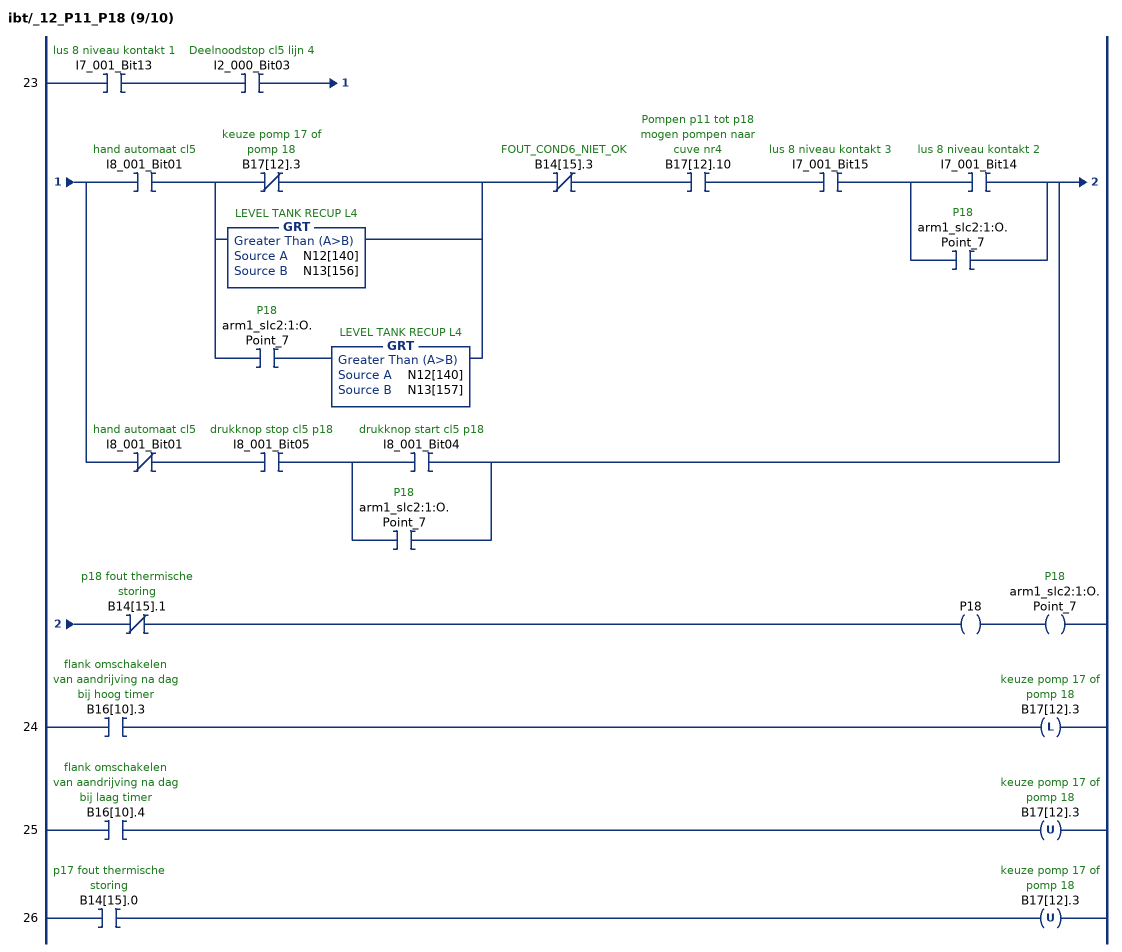
   23: XIC(I7_001_Bit13)XIC(I2_000_Bit03)[XIC(I8_001_Bit01) [XIO(B17[12].3) ,GRT(N12[140],N13[156]) ,XIC(arm1_slc2:1:O.Point_7) GRT(N12[140],N13[157]) ] XIO(B14[15].3) XIC(B17[12].10) XIC(I7_001_Bit15) [XIC(I7_001_Bit14) ,XIC(arm1_slc2:1:O.Point_7) ] ,XIO(I8_001_Bit01) XIC(I8_001_Bit05) [XIC(I8_001_Bit04) ,XIC(arm1_slc2:1:O.Point_7) ] ]XIO(B14[15].1)OTE(P18)OTE(arm1_slc2:1:O.Point_7);
   24: XIC(B16[10].3)OTL(B17[12].3);
   25: XIC(B16[10].4)OTU(B17[12].3);
   26: XIC(B14[15].0)OTU(B17[12].3);
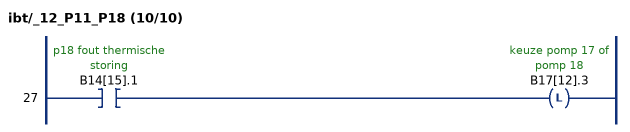
   27: XIC(B14[15].1)OTL(B17[12].3);
END_ROUTINE
